RoboDK station: deburrBot.rdk

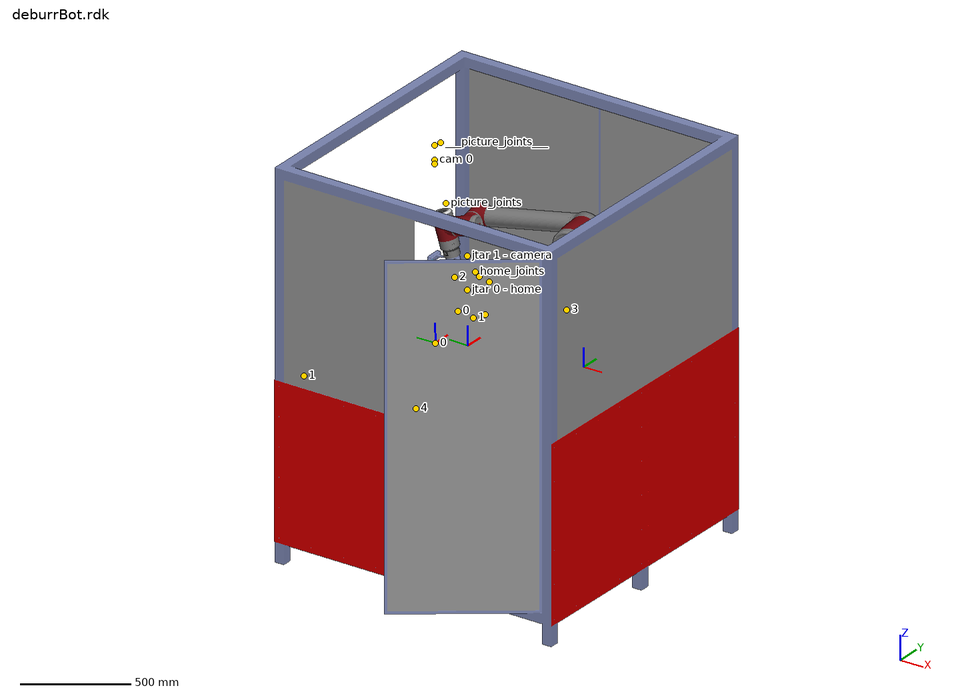
[picture v0: the station drawn from its stored meshes, robots at their saved joint values, targets as dots, program paths as lines]
Station deburrBot (saved by RoboDK 5.5.3). Poses are relative to the parent item; angles as X-Y-Z fixed-axis rotations.
  - frame world at (0, 0, 0) mm
    - folder robot
      - robot jaka12 (model Jaka Zu12): 6 axes, payload 12 kg, reach 1327 mm, repeatability 0.03 mm, weight 41 kg
          modified DH rows (alpha deg, a mm, theta deg, d mm): 0, 0, 180, 142.65; 90, 0, 0, 0; 0, 595, 0, 0; 0, 571.5, -180, -131.5; -90, 0, 0, 115; 90, 0, 180, 103.5
          base shift (0, 0, 0) mm, rotated rx 0 ry 0 rz 180 deg
          joint limits [-360, -85, -175, -85, -360, -360] to [360, 265, 175, 265, 360, 360]; home [180.17, 108.14, -152.76, 226.01, 89.5, -165.58]; saved at [-170.709, 94.649, -102.296, 82.411, 91.833, 217.942]
        - tool zero, TCP at (0, 0, 0) mm
        - tool WC Angle Grinder Tool Assy 00 w Camera, TCP at (-139.39, 64.58, 199.93) mm, rotated rx -169.95 ry 0.29 rz -115.89 deg, size 183.8 x 204.5 x 380.3 mm, geometry from WC Angle Grinder Tool Assy 00 w Camera.STEP
        - tool camera tcp, TCP at (78.21, 73.4, 50.54) mm, rotated rx 15.29 ry -0.46 rz 150.04 deg
        - tool temp_rdk_gen_tool, TCP at (119.73, 140.78, 339.91) mm, rotated rx -164.71 ry -0.46 rz 150.04 deg
    - folder Joints
      - target home_joints (joint target) at (-610.5, 21.02, 299.9) mm, rotated rx -0.18 ry 0 rz 91.08 deg; joints [-197.245, 108.097, -114.41, 86.508, 87.072, 97.84] of jaka12
      - target ___picture_joints___ (joint target) at (-788.33, 3.1, 904.1) mm, rotated rx -0.18 ry 0 rz 91.08 deg; joints [-193.281, 70.189, -24.921, 29.93, 85.912, 196.146] of jaka12
      - target picture_joints (joint target) at (-788.08, 43.13, 584.1) mm, rotated rx -0.18 ry 0 rz 91.08 deg; joints [-196.357, 72.51, -31.124, 34.045, 85.132, 193.161] of jaka12
      - target temp1_picture_joints__ (joint target) at (-669.95, 215.41, 154.49) mm, rotated rx -0.18 ry 0 rz 91.08 deg; joints [-213.749, 93.236, -101.522, 85.785, 81.031, 176.131] of jaka12
      - target temp2_picture_joints__ (joint target) at (-522.51, -74.1, 337.62) mm, rotated rx 10.34 ry -15.34 rz 1.06 deg; joints [-170.709, 94.649, -102.296, 82.411, 91.833, 217.942] of jaka12
    - frame workstation at (-809.08, -11.32, -100.97) mm, rotated rx -0.18 ry 0 rz 91.08 deg
      - frame working area at (0, 0, 0) mm
        - target 0 (Cartesian target) at (0, 0, 0) mm; joints [-190.737, 67.653, -119.383, 131.902, 88.146, 109.423] of jaka12
        - target 1 (Cartesian target) at (-610, 305, 0) mm; joints [-155.286, 29.029, -48.291, 100.162, 94.163, 144.382] of jaka12
        - target 2 (Cartesian target) at (610, 305, 0) mm; joints [-217.503, 28.973, -48.423, 101.486, 83.931, 82.919] of jaka12
        - target 3 (Cartesian target) at (610, -305, 0) mm; joints [-247.067, 65.086, -116.99, 137.973, 80.798, 53.249] of jaka12
        - target 4 (Cartesian target) at (-610, -305, 0) mm; joints [-133.69, 65.557, -116.818, 134.317, 97.213, 165.872] of jaka12
        - frame camera at (0, 0, 0) mm
          - target cam 0 (joint target) at (0, 0, 919.4) mm; joints [-190.779, 75.86, -36.332, 25.86, 85.467, 20.21] of jaka12
          - target cam 1 (joint target) at (0, 0, 900) mm; joints [-192.076, 79.927, -35.831, 16.455, 83.995, 109.503] of jaka12
          - target cam 2 (joint target) at (0, 0, 992.72) mm; joints [-190.304, 75.984, -40.965, 40.212, 87.347, 200.04] of jaka12
      - frame eye in hand calibration at (0, 0, 0) mm
        - target 0 (Cartesian target) at (0, 0, 0) mm; joints [-190.737, 67.653, -119.383, 131.902, 88.146, 109.423] of jaka12
        - target 1 (Cartesian target) at (0, 0, 0) mm, rotated rx 30 ry 0 rz 0 deg; joints [-197.704, 75.955, -138.557, 166.921, 94.514, 192.863] of jaka12
    - frame desk_workstation at (-675, 50, -100) mm, rotated rx 0 ry 0 rz 90 deg
      - frame desk_jtars at (0, 0, 0) mm
        - target jtar 0 - home (joint target) at (0, 0, 280) mm; joints [-198.106, 98.017, -119.274, 101.743, 86.906, 102.151] of jaka12
        - target jtar 1 - camera (joint target) at (0, 0, 450) mm, rotated rx 180 ry 0 rz 0 deg; joints [-200.006, 95.084, -113.084, 93.868, 84.92, 190.624] of jaka12
        - target jtar 2 - testing force moves (joint target) at (140, 0, 100) mm; joints [-210.775, 84.006, -127.25, 124.63, 84.903, 89.609] of jaka12
      - frame finish_force_taget_run_fn at (0, 0, 0) mm
        - target 0 (Cartesian target) at (180, 180, 50) mm; joints [-206.499, 65.378, -108.411, 124.065, 85.556, 93.849] of jaka12
        - target 1 (Cartesian target) at (160, 80, 50) mm; joints [-208.755, 73.052, -120.147, 128.307, 85.208, 91.613] of jaka12
    - frame 3D at (0, 0, 0) mm
      - object Station Assy 00 rdk 3D at (0, 0, 0) mm, size 1328.1 x 1222.2 x 1371.6 mm, geometry from Station Assy 00 rdk 3D.STEP
      - object RH2 frame grinder at (0, 0, 0) mm, size 1473.2 x 1981.2 x 1532.7 mm, geometry from RH2 frame grinder.STEP
      - object RH2 ROBOT JAKA at (0, 0, 0) mm, size 1891.7 x 1981.2 x 1527 mm, geometry from RH2 ROBOT JAKA.STEP
